(* Logix 5000 project; controller R5_CSS vendor 1 type 14 code 74 rev 19.11; software revision 19.01; part 3 of 20 *)
(* tags used below, declared in another part *)
   AT102A_SCP : SCLP;   // QUENCH WATER CONDUCTIVITY TRANSMITTER SCALER (0-100 milli Siemens)
   AC102A : ANALYTICAL;   // QUENCH WATER CONDUCTIVITY CONTROL
   AlarmMaster : DINT;
   Coal_Tank_Heel_Inches : REAL;
   FC215 : FLOW_CONTROL;   // OVERHEAD CONDENSER CHILLED WATER FLOW CONTROL
   FC365 : FLOW_CONTROL;   // COALESCER PROCESS IMPURITY FLOW CONTROL
   FC370 : FLOW_CONTROL;   // COALESCER MAKE UP WATER FLOW CONTROL
   FC406 : FLOW_CONTROL;   // HX COOLING WATER FLOW CONTROL
   FC_215SCP : SCLP;   // OVERHEAD CONDENSER CHILLED WATER FLOW TRANSMITTER SCALER
   FC_406SCP : SCLP;   // HX COOLING WATER FLOW TRANMITTER SCALER
   FCV410_Open : BOOL;
   FIT08 : BOOL;
   FIT101 : BOOL;
   FIT140A : BOOL;
   FIT140B : BOOL;
   FIT365_SCP : SCLP;   // COALESCER PROCESS IMPURITY FLOW
   FIT370_SCP : SCLP;   // COALESCER MAKE UP WATER SCALER
   FIT403 : BOOL;
   HCP_FAULT : BOOL;
   HS104A : ValveControl_TwoWay;
   HS104B : ValveControl_TwoWay;
   HS141 : ValveControl_TwoWay;
   HS315A : ValveControl_TwoWay;
   HS315B : ValveControl_TwoWay;
   HS431A : ValveControl_TwoWay;
   HS431B : ValveControl_TwoWay;
   HS433A : ValveControl_TwoWay;
   HS433B : ValveControl_TwoWay;
   HT_FAULT : BOOL;
   HTGA : BOOL;
   HX401A : PUMP_CONTROL;   // HEAT EXCHANGER A
   HX401B : PUMP_CONTROL;   // HEAT EXCHANGER B
   InputMax_IF8 : REAL;
   InputMin_IF8 : REAL;
   LC205 : LEVEL_CONTROL;   // OVERHEAD CONDENSER BASIN LEVEL CONTROL
   LC302 : LEVEL_CONTROL;   // COALESCER OIL CHAMBER LEVEL CONTROL
   LC302_LT_Raw : REAL;
   LC302_SP : SCLP;   // COALESCER OIL CHAMBER LEVEL TRANSMITTER SCALER
   LC_205_SCP : SCLP;   // OVERHEAD CONDENSER BASIN LEVEL TRANSMITTER SCALER
   LossOfSignal_mA : DINT;
   MV361_Open : BOOL;
   P101A : PUMP_CONTROL;
   P101B : PUMP_CONTROL;
   P205 : PUMP_CONTROL;   // OVERHEAD CONDENSER TRANSFER PUMP
   P302A : PUMP_CONTROL;
   P302B : PUMP_CONTROL;
   P303A : PUMP_CONTROL;
   P303B : PUMP_CONTROL;
   PC101A : PRESSURE_CONTROL;   // LOWER QUENCH TOWER PRESSURE TRANSMITTER
   PC101B : PRESSURE_CONTROL;   // UPPER QUENCH TOWER PRESSURE TRANSMITTER PRESSURE CONTOL
   PC102A : PRESSURE_CONTROL;   // QUENCH BASIN TRANSFER PUMP SUCTION PRESSURE CONTROL
   PC102B : PRESSURE_CONTROL;   // QUENCH BASIN TRANSFER PUMP DISCHARGE PRESSURE CONTROL
   PC214 : PRESSURE_CONTROL;   // VACUUM SYSTEM PRESSURE TRANSMITTER
   PC214_PID_PV_Select : DINT;   // 0 = PT214 1 = PT101A 2 = PT101B
   PC214_SCP : SCLP;   // VACUUM SYSTEM PRESSURE TRANSMITTER SCALER
   PC271 : PRESSURE_CONTROL;   // VENT HEADER PRESSURE CONTROL
   PC407A : PRESSURE_CONTROL;   // PRE HX LOW PRESSURE TRANSMITTER
   PC407B : PRESSURE_CONTROL;   // POST HX LOW PRESSURE TRANSMITTER
   PIT101A_SCP : SCLP;   // LOWER QUENCH TOWER PRESSURE TRANSMITTER SCALER
   PIT101B_SCP : SCLP;   // UPPER QUENCH TOWER PRESSURE TRANSMITTER SCALER
   PIT102A_SCP : SCLP;   // QUENCH BASIN TRANSFER PUMP SUCTION PRESSURE INDICATOR SCALER
   PIT102B_SCP : SCLP;   // QUENCH BASIN TRANSFER PUMP DISCHARGE PRESSURE SCALER
   PIT407A_SCP : SCLP;   // PRE HX LOW PRESSURE TRANSMITTER
   PIT407B_SCP : SCLP;   // POST HX LOW PRESSURE TRANSMITTER SCALER
   PT271_SCP : SCLP;   // VENT HEADER PRESSURE TRANSMITTER SCALER
   SignalLossHigh_IF8 : DINT;
   SignalLossLow_IF8 : DINT;
   TAS15569 : BOOL;
   TC108 : TEMP_CONTROL;   // QUENCH TOWER EXIT GAS TEMPERATURE CONTROL
   TC114A : TEMP_CONTROL;   // QUENCH BASIN SHELL TEMPERATURE CONTROL
   TC114B : TEMP_CONTROL;   // QUENCH BASIN LIQUID TEMPERATURE CONTROL
   TC121A : TEMP_CONTROL;   // GTL FROM PRUA TEMPERATURE CONTROL
   TC121B : TEMP_CONTROL;   // GTL FROM PRUB TEMPERATURE CONTROL
   TC121C : TEMP_CONTROL;   // GTL FROM PRUC TEMPERATURE CONTROL
   TC121D : TEMP_CONTROL;   // GTL FROM PRUD TEMPERATURE CONTROL
   TC121E : TEMP_CONTROL;
   TC121F : TEMP_CONTROL;
   TC121G : TEMP_CONTROL;
   TC121H : TEMP_CONTROL;
   TC123A : TEMP_CONTROL;   // HEAT JACKET VENT FROM PRUA TEMPERATURE CONTROL
   TC123A_SCP : SCLP;   // HEAT JACKET VENT FROM PRUA TEMPERATURE TRANSMITTER SCALER
   TC123B : TEMP_CONTROL;
   TC123B_SCP : SCLP;   // HEAT JACKET VENT FROM PRUB TEMPERATURE TRANSMITTER SCALER
   TC123C : TEMP_CONTROL;   // HEAT JACKET VENT FROM PRUC TEMPERATURE CONTROL
   TC123C_SCP : SCLP;   // HEAT JACKET VENT FROM PRUC TEMPERATURE TRANSMITTER SCALER
   TC123D : TEMP_CONTROL;   // HEAT JACKET VENT FROM PRUD TEMPERATURE TRANSMITTER
   TC123D_SCP : SCLP;   // HEAT JACKET VENT FROM PRUD TEMPERATURE TRANSMITTER SCALER
   TC123E : TEMP_CONTROL;
   TC123E_SCP : SCLP;
   TC123F : TEMP_CONTROL;
   TC123F_SCP : SCLP;
   TC123G : TEMP_CONTROL;
   TC123G_SCP : SCLP;
   TC306 : TEMP_CONTROL;
   TC313A : TEMP_CONTROL;   // PRIMARY COALESCER SEPARATOR TEMPERATURE CONTROL
   TC319 : TEMP_CONTROL;   // COALESCER OIL CHAMBER PROCESS TEMPERATURE CONTROL
   TT108_SCP : SCLP;   // QUENCH TOWER EXIT GAS TEMPERATURE TRANSMITTER SCALER
   TT121A_SCP : SCLP;   // GTL FROM PRUA TEMPERATURE TRANSMITTER SCALER
   TT121B_SCP : SCLP;
   TT121C_SCP : SCLP;
   TT121D_SCP : SCLP;
   TT121E_SCP : SCLP;
   TT121F_SCP : SCLP;   // GTL FROM PRUB TEMPERATURE TRANSMITTER SCALER
   TT121G_SCP : SCLP;   // GTL FROM PRUC TEMPERATURE TRANSMITTER SCALER
   TT121H_SCP : SCLP;   // GTL FROM PRUD TEMPERATURE TRANSMITTER SCALER
(* MainProgram, continued *)

ROUTINE A1c_MDI   (* ladder *)
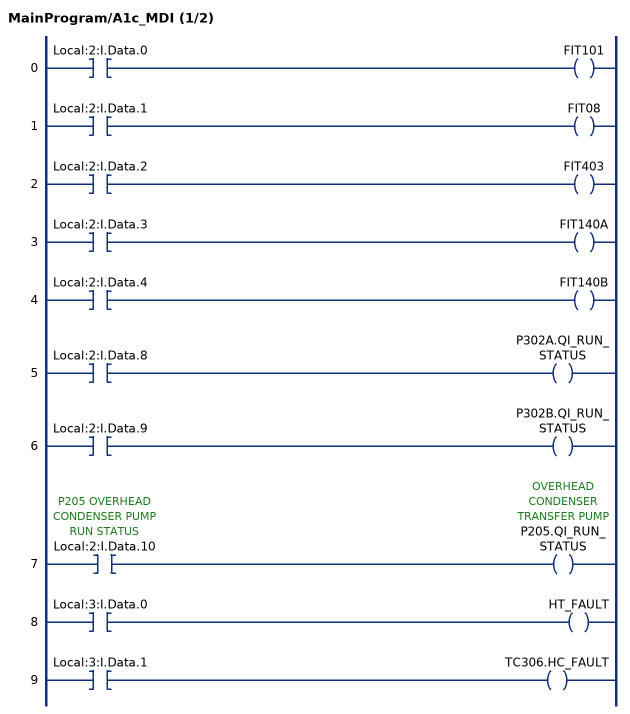
   0: XIC(Local:2:I.Data.0)OTE(FIT101);
   1: XIC(Local:2:I.Data.1)OTE(FIT08);
   2: XIC(Local:2:I.Data.2)OTE(FIT403);
   3: XIC(Local:2:I.Data.3)OTE(FIT140A);
   4: XIC(Local:2:I.Data.4)OTE(FIT140B);
   5: XIC(Local:2:I.Data.8)OTE(P302A.QI_RUN_STATUS);
   6: XIC(Local:2:I.Data.9)OTE(P302B.QI_RUN_STATUS);
   7: XIC(Local:2:I.Data.10)OTE(P205.QI_RUN_STATUS);
   8: XIC(Local:3:I.Data.0)OTE(HT_FAULT);
   9: XIC(Local:3:I.Data.1)OTE(TC306.HC_FAULT);
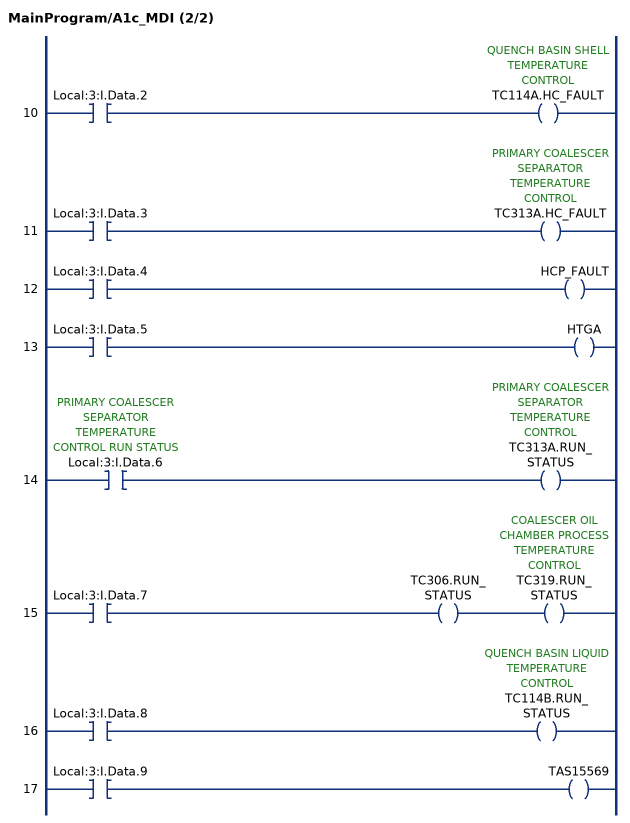
   10: XIC(Local:3:I.Data.2)OTE(TC114A.HC_FAULT);
   11: XIC(Local:3:I.Data.3)OTE(TC313A.HC_FAULT);
   12: XIC(Local:3:I.Data.4)OTE(HCP_FAULT);
   13: XIC(Local:3:I.Data.5)OTE(HTGA);
   14: XIC(Local:3:I.Data.6)OTE(TC313A.RUN_STATUS);
   15: XIC(Local:3:I.Data.7)OTE(TC306.RUN_STATUS)OTE(TC319.RUN_STATUS);
   16: XIC(Local:3:I.Data.8)OTE(TC114B.RUN_STATUS);
   17: XIC(Local:3:I.Data.9)OTE(TAS15569);
END_ROUTINE

ROUTINE A1d_MDO   (* ladder *)
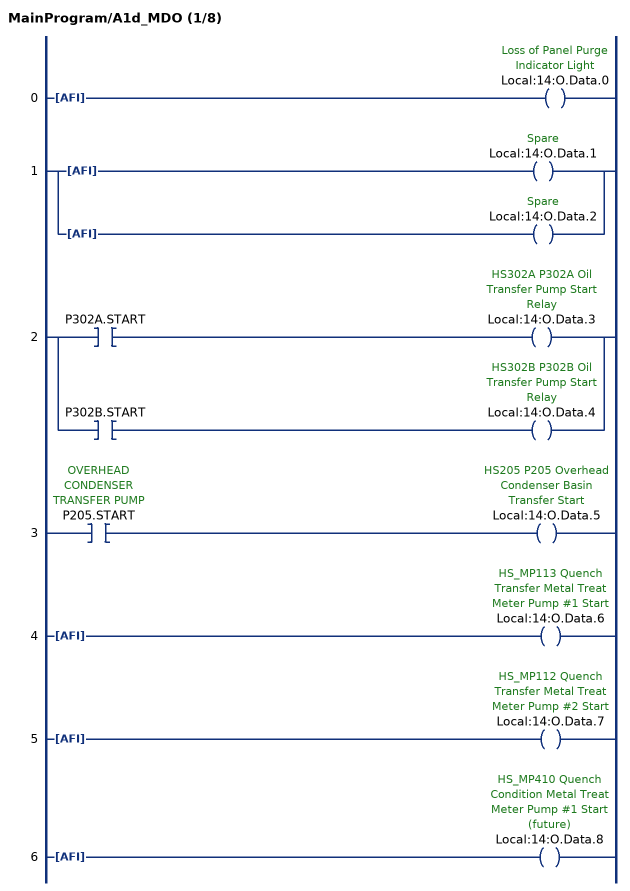
   0: AFI()OTE(Local:14:O.Data.0);
   1: [AFI() OTE(Local:14:O.Data.1) ,AFI() OTE(Local:14:O.Data.2) ];
   2: [XIC(P302A.START) OTE(Local:14:O.Data.3) ,XIC(P302B.START) OTE(Local:14:O.Data.4) ];
   3: XIC(P205.START)OTE(Local:14:O.Data.5);
   4: AFI()OTE(Local:14:O.Data.6);
   5: AFI()OTE(Local:14:O.Data.7);
   6: AFI()OTE(Local:14:O.Data.8);
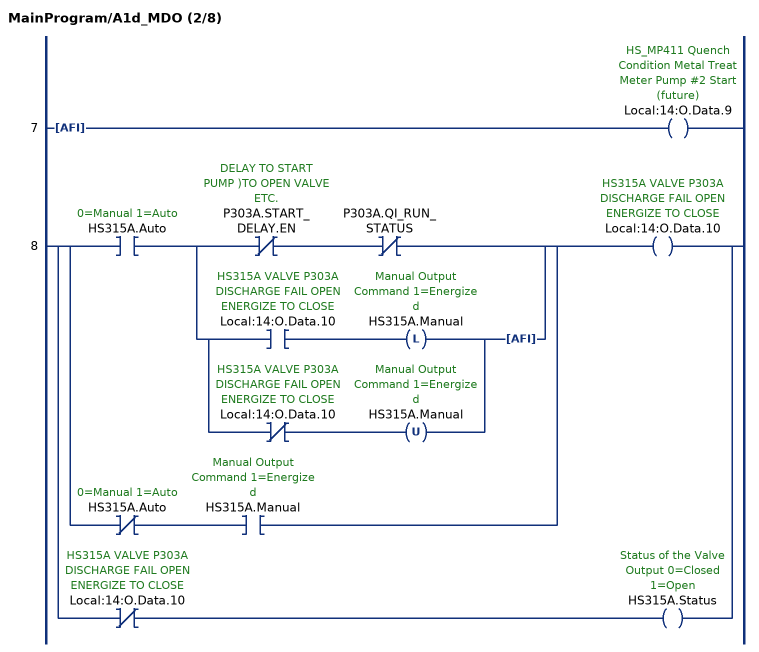
   7: AFI()OTE(Local:14:O.Data.9);
   8: [[XIC(HS315A.Auto) [XIO(P303A.START_DELAY.EN) XIO(P303A.QI_RUN_STATUS) ,[XIC(Local:14:O.Data.10) OTL(HS315A.Manual) ,XIO(Local:14:O.Data.10) OTU(HS315A.Manual) ] AFI() ] ,XIO(HS315A.Auto) XIC(HS315A.Manual) ] OTE(Local:14:O.Data.10) ,XIO(Local:14:O.Data.10) OTE(HS315A.Status) ];
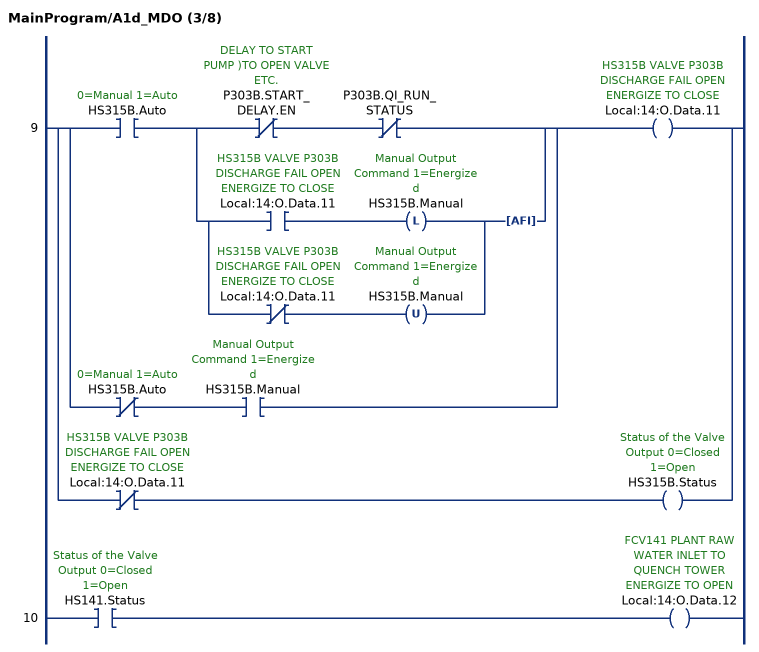
   9: [[XIC(HS315B.Auto) [XIO(P303B.START_DELAY.EN) XIO(P303B.QI_RUN_STATUS) ,[XIC(Local:14:O.Data.11) OTL(HS315B.Manual) ,XIO(Local:14:O.Data.11) OTU(HS315B.Manual) ] AFI() ] ,XIO(HS315B.Auto) XIC(HS315B.Manual) ] OTE(Local:14:O.Data.11) ,XIO(Local:14:O.Data.11) OTE(HS315B.Status) ];
   10: XIC(HS141.Status)OTE(Local:14:O.Data.12);
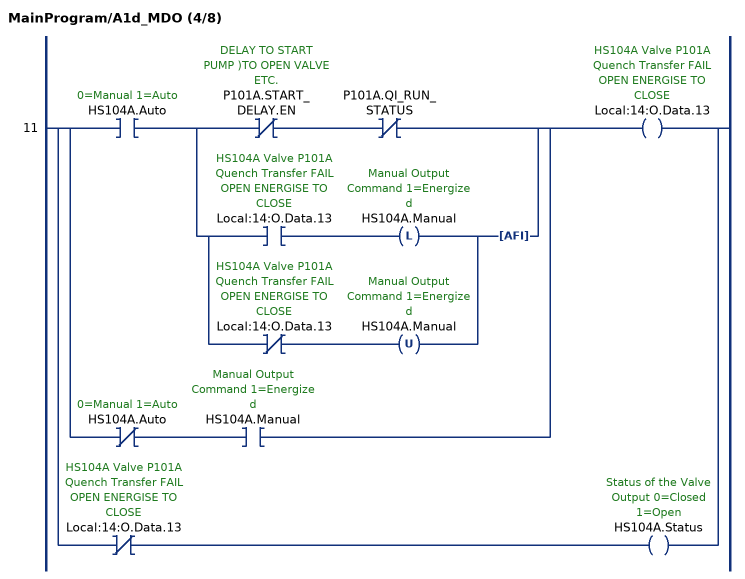
   11: [[XIC(HS104A.Auto) [XIO(P101A.START_DELAY.EN) XIO(P101A.QI_RUN_STATUS) ,[XIC(Local:14:O.Data.13) OTL(HS104A.Manual) ,XIO(Local:14:O.Data.13) OTU(HS104A.Manual) ] AFI() ] ,XIO(HS104A.Auto) XIC(HS104A.Manual) ] OTE(Local:14:O.Data.13) ,XIO(Local:14:O.Data.13) OTE(HS104A.Status) ];
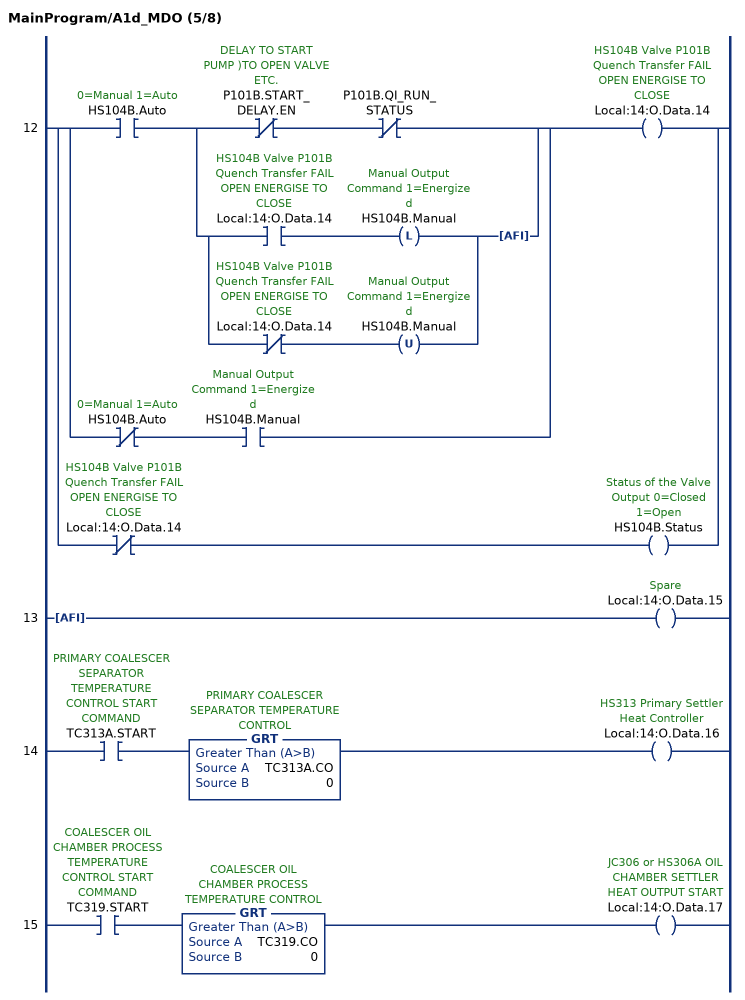
   12: [[XIC(HS104B.Auto) [XIO(P101B.START_DELAY.EN) XIO(P101B.QI_RUN_STATUS) ,[XIC(Local:14:O.Data.14) OTL(HS104B.Manual) ,XIO(Local:14:O.Data.14) OTU(HS104B.Manual) ] AFI() ] ,XIO(HS104B.Auto) XIC(HS104B.Manual) ] OTE(Local:14:O.Data.14) ,XIO(Local:14:O.Data.14) OTE(HS104B.Status) ];
   13: AFI()OTE(Local:14:O.Data.15);
   14: XIC(TC313A.START)GRT(TC313A.CO,0)OTE(Local:14:O.Data.16);
   15: XIC(TC319.START)GRT(TC319.CO,0)OTE(Local:14:O.Data.17);
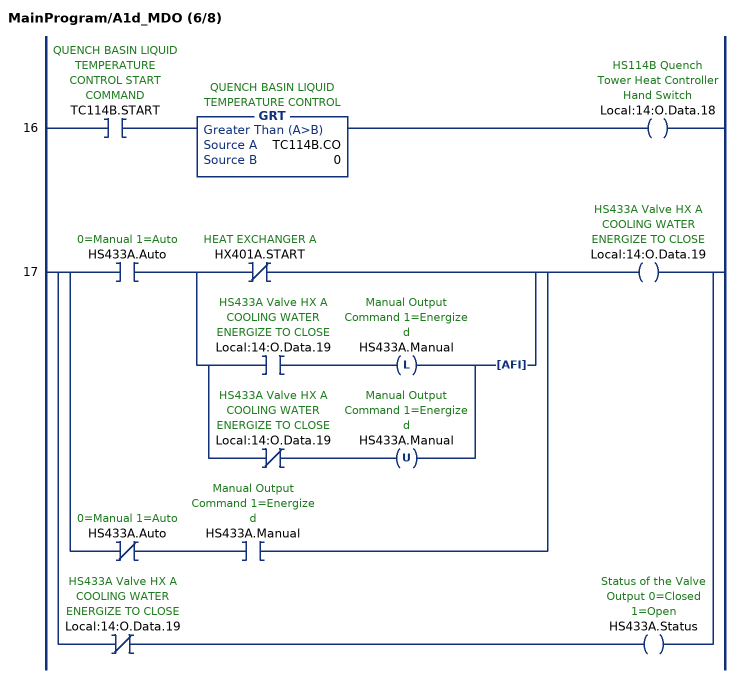
   16: XIC(TC114B.START)GRT(TC114B.CO,0)OTE(Local:14:O.Data.18);
   17: [[XIC(HS433A.Auto) [XIO(HX401A.START) ,[XIC(Local:14:O.Data.19) OTL(HS433A.Manual) ,XIO(Local:14:O.Data.19) OTU(HS433A.Manual) ] AFI() ] ,XIO(HS433A.Auto) XIC(HS433A.Manual) ] OTE(Local:14:O.Data.19) ,XIO(Local:14:O.Data.19) OTE(HS433A.Status) ];
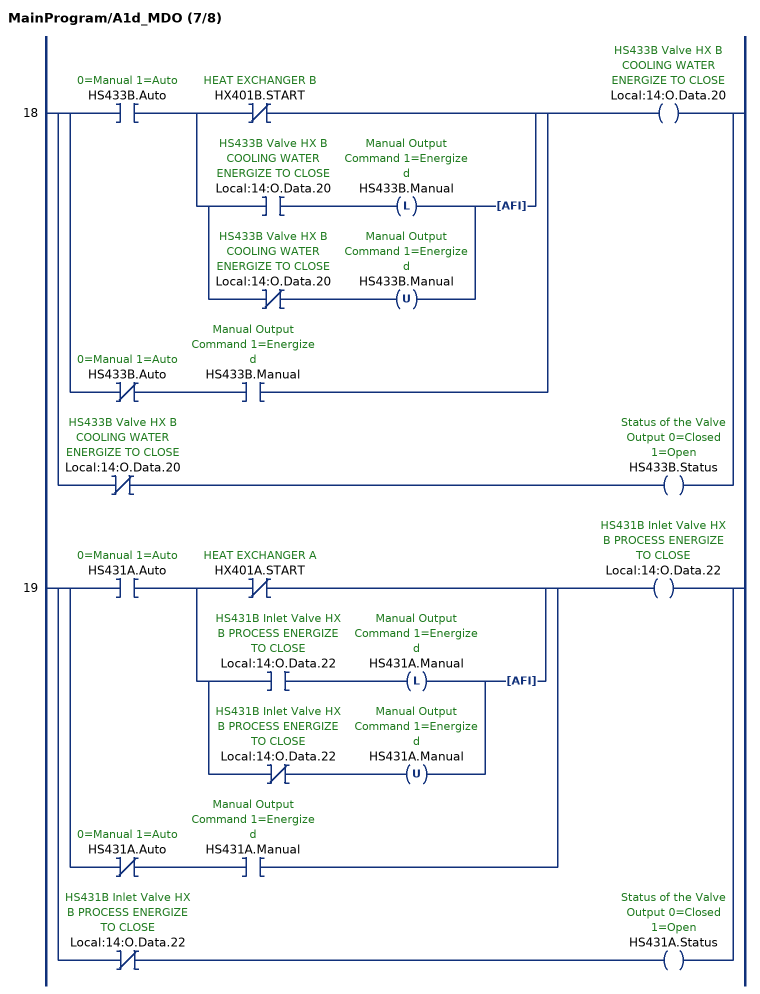
   18: [[XIC(HS433B.Auto) [XIO(HX401B.START) ,[XIC(Local:14:O.Data.20) OTL(HS433B.Manual) ,XIO(Local:14:O.Data.20) OTU(HS433B.Manual) ] AFI() ] ,XIO(HS433B.Auto) XIC(HS433B.Manual) ] OTE(Local:14:O.Data.20) ,XIO(Local:14:O.Data.20) OTE(HS433B.Status) ];
   19: [[XIC(HS431A.Auto) [XIO(HX401A.START) ,[XIC(Local:14:O.Data.22) OTL(HS431A.Manual) ,XIO(Local:14:O.Data.22) OTU(HS431A.Manual) ] AFI() ] ,XIO(HS431A.Auto) XIC(HS431A.Manual) ] OTE(Local:14:O.Data.22) ,XIO(Local:14:O.Data.22) OTE(HS431A.Status) ];
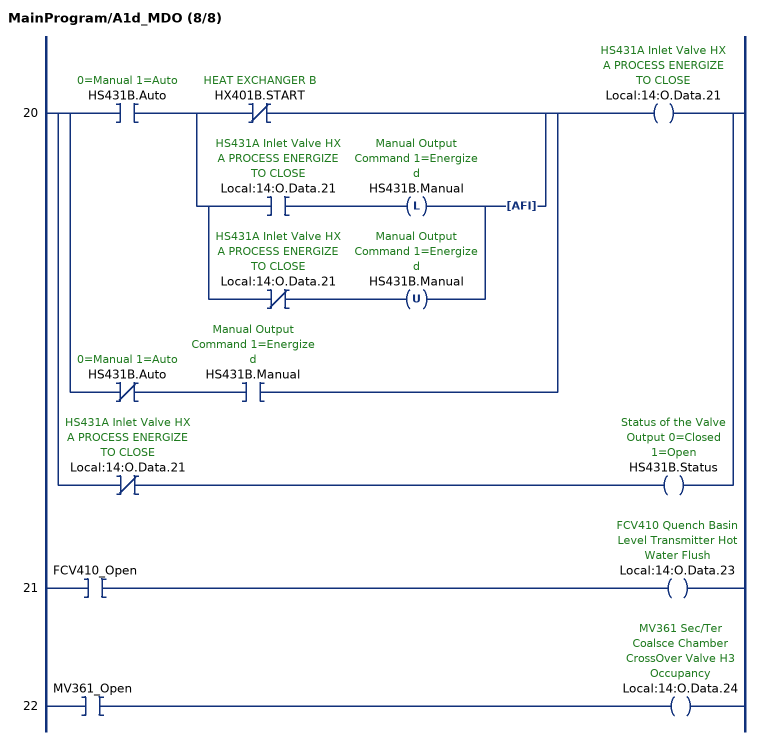
   20: [[XIC(HS431B.Auto) [XIO(HX401B.START) ,[XIC(Local:14:O.Data.21) OTL(HS431B.Manual) ,XIO(Local:14:O.Data.21) OTU(HS431B.Manual) ] AFI() ] ,XIO(HS431B.Auto) XIC(HS431B.Manual) ] OTE(Local:14:O.Data.21) ,XIO(Local:14:O.Data.21) OTE(HS431B.Status) ];
   21: XIC(FCV410_Open)OTE(Local:14:O.Data.23);
   22: XIC(MV361_Open)OTE(Local:14:O.Data.24);
END_ROUTINE

ROUTINE A1e_MAI_SCP   (* ladder *)
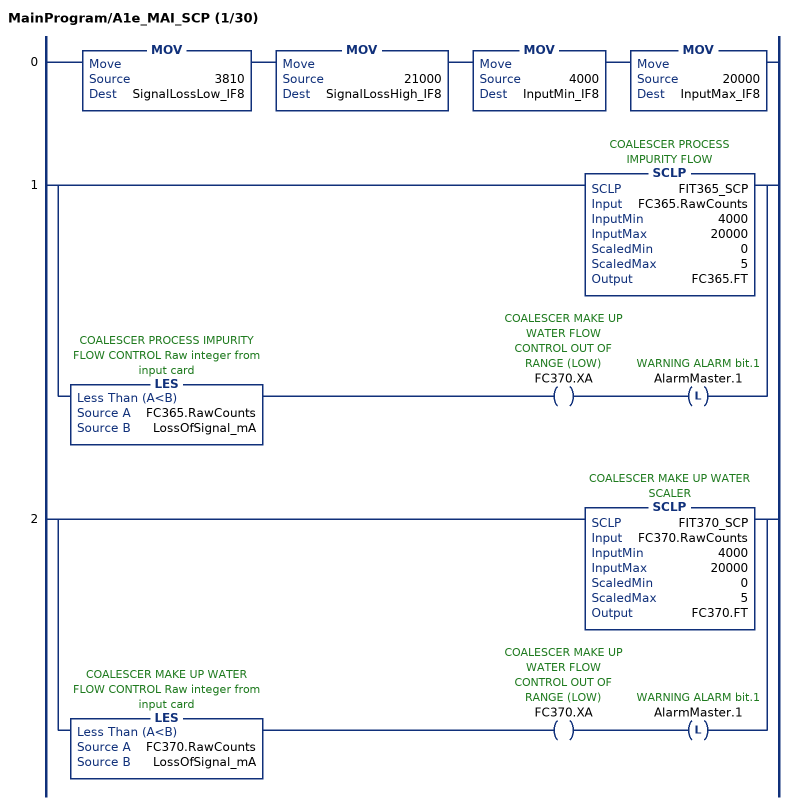
   0: MOV(3810,SignalLossLow_IF8)MOV(21000,SignalLossHigh_IF8)MOV(4000,InputMin_IF8)MOV(20000,InputMax_IF8);
   1: [SCLP(FIT365_SCP,FC365.RawCounts,4000,20000,0,5,FC365.FT) ,LES(FC365.RawCounts,LossOfSignal_mA) OTE(FC370.XA) OTL(AlarmMaster.1) ];
   2: [SCLP(FIT370_SCP,FC370.RawCounts,4000,20000,0,5,FC370.FT) ,LES(FC370.RawCounts,LossOfSignal_mA) OTE(FC370.XA) OTL(AlarmMaster.1) ];
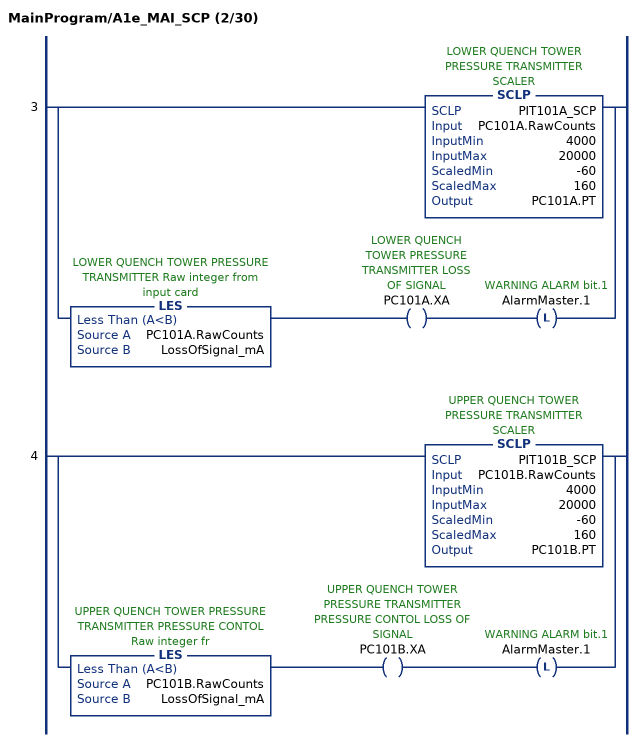
   3: [SCLP(PIT101A_SCP,PC101A.RawCounts,4000,20000,-60,160,PC101A.PT) ,LES(PC101A.RawCounts,LossOfSignal_mA) OTE(PC101A.XA) OTL(AlarmMaster.1) ];
   4: [SCLP(PIT101B_SCP,PC101B.RawCounts,4000,20000,-60,160,PC101B.PT) ,LES(PC101B.RawCounts,LossOfSignal_mA) OTE(PC101B.XA) OTL(AlarmMaster.1) ];
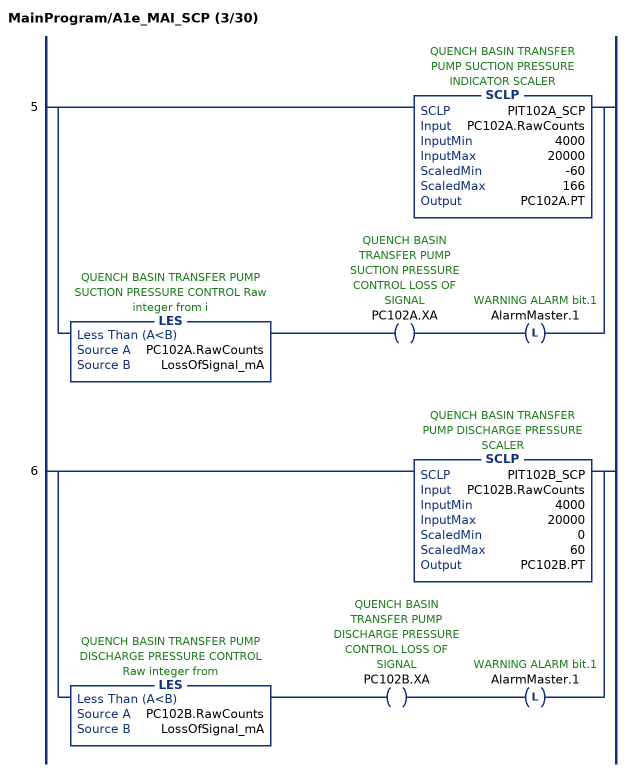
   5: [SCLP(PIT102A_SCP,PC102A.RawCounts,4000,20000,-60,166,PC102A.PT) ,LES(PC102A.RawCounts,LossOfSignal_mA) OTE(PC102A.XA) OTL(AlarmMaster.1) ];
   6: [SCLP(PIT102B_SCP,PC102B.RawCounts,4000,20000,0,60,PC102B.PT) ,LES(PC102B.RawCounts,LossOfSignal_mA) OTE(PC102B.XA) OTL(AlarmMaster.1) ];
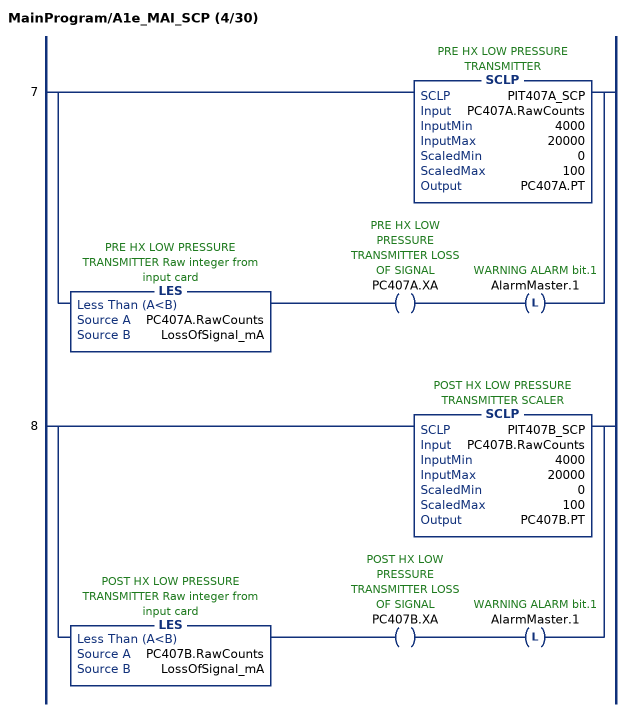
   7: [SCLP(PIT407A_SCP,PC407A.RawCounts,4000,20000,0,100,PC407A.PT) ,LES(PC407A.RawCounts,LossOfSignal_mA) OTE(PC407A.XA) OTL(AlarmMaster.1) ];
   8: [SCLP(PIT407B_SCP,PC407B.RawCounts,4000,20000,0,100,PC407B.PT) ,LES(PC407B.RawCounts,LossOfSignal_mA) OTE(PC407B.XA) OTL(AlarmMaster.1) ];
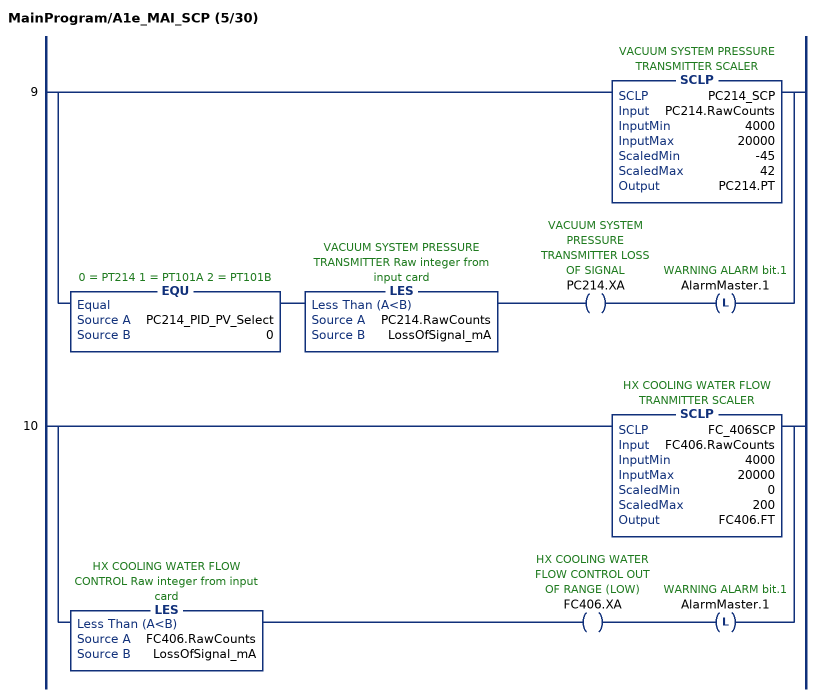
   9: [SCLP(PC214_SCP,PC214.RawCounts,4000,20000,-45,42,PC214.PT) ,EQU(PC214_PID_PV_Select,0) LES(PC214.RawCounts,LossOfSignal_mA) OTE(PC214.XA) OTL(AlarmMaster.1) ];
   10: [SCLP(FC_406SCP,FC406.RawCounts,4000,20000,0,200,FC406.FT) ,LES(FC406.RawCounts,LossOfSignal_mA) OTE(FC406.XA) OTL(AlarmMaster.1) ];
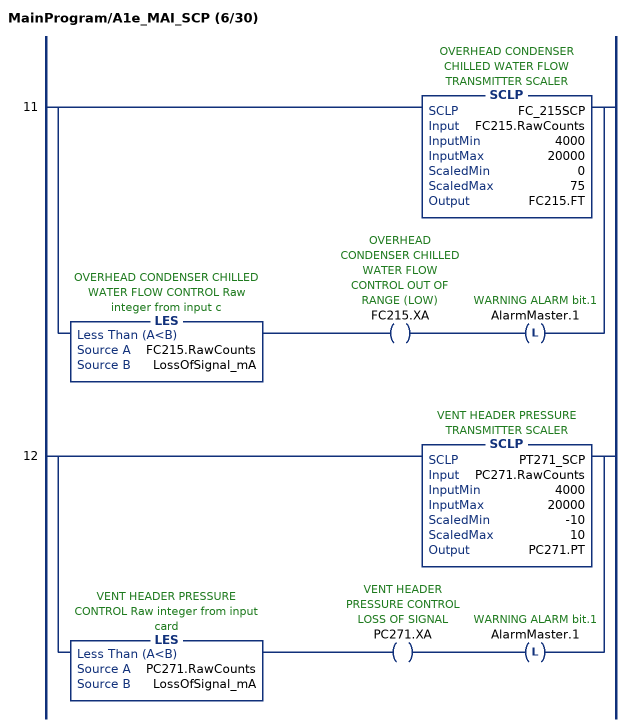
   11: [SCLP(FC_215SCP,FC215.RawCounts,4000,20000,0,75,FC215.FT) ,LES(FC215.RawCounts,LossOfSignal_mA) OTE(FC215.XA) OTL(AlarmMaster.1) ];
   12: [SCLP(PT271_SCP,PC271.RawCounts,4000,20000,-10,10,PC271.PT) ,LES(PC271.RawCounts,LossOfSignal_mA) OTE(PC271.XA) OTL(AlarmMaster.1) ];
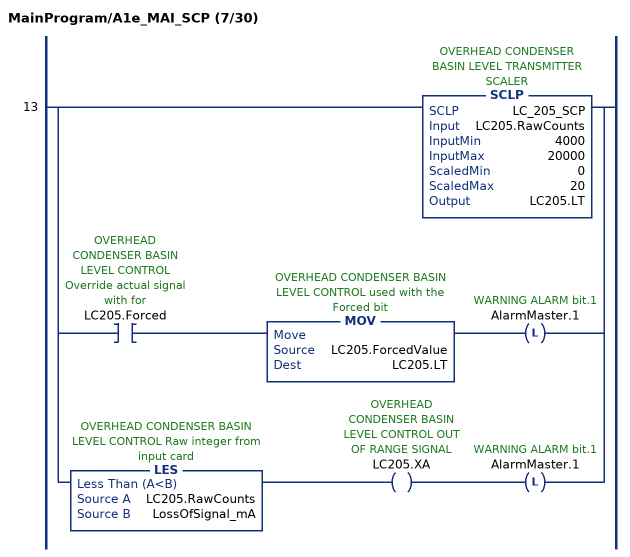
   13: [SCLP(LC_205_SCP,LC205.RawCounts,4000,20000,0,20,LC205.LT) ,XIC(LC205.Forced) MOV(LC205.ForcedValue,LC205.LT) OTL(AlarmMaster.1) ,LES(LC205.RawCounts,LossOfSignal_mA) OTE(LC205.XA) OTL(AlarmMaster.1) ];
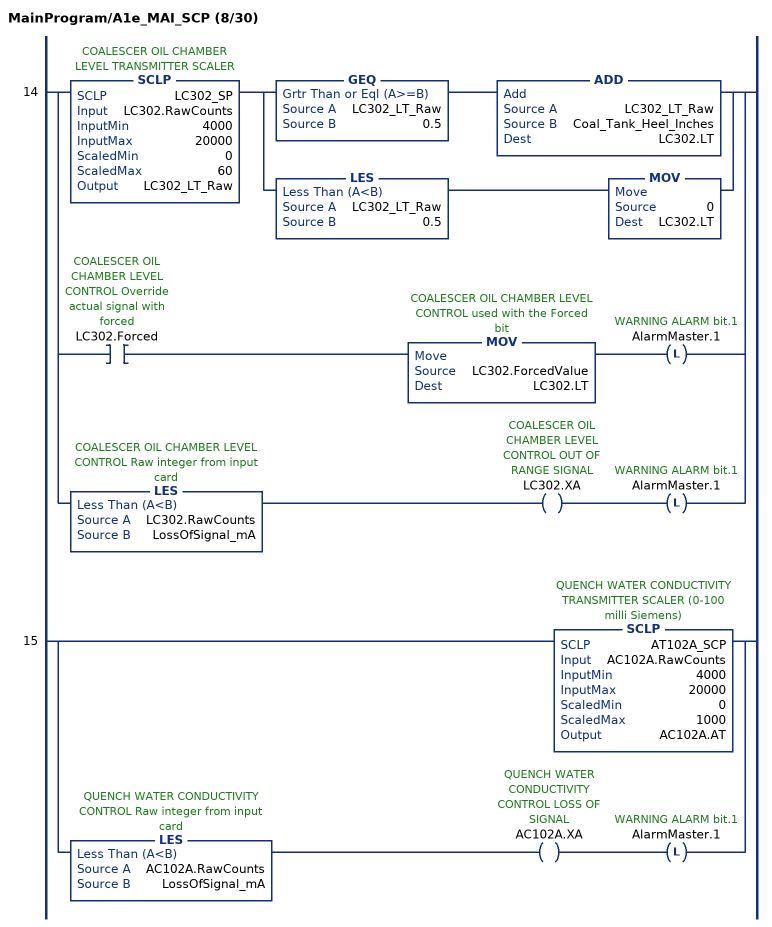
   14: [SCLP(LC302_SP,LC302.RawCounts,4000,20000,0,60,LC302_LT_Raw) [GEQ(LC302_LT_Raw,0.5) ADD(LC302_LT_Raw,Coal_Tank_Heel_Inches,LC302.LT) ,LES(LC302_LT_Raw,0.5) MOV(0,LC302.LT) ] ,XIC(LC302.Forced) MOV(LC302.ForcedValue,LC302.LT) OTL(AlarmMaster.1) ,LES(LC302.RawCounts,LossOfSignal_mA) OTE(LC302.XA) OTL(AlarmMaster.1) ];
   15: [SCLP(AT102A_SCP,AC102A.RawCounts,4000,20000,0,1000,AC102A.AT) ,LES(AC102A.RawCounts,LossOfSignal_mA) OTE(AC102A.XA) OTL(AlarmMaster.1) ];
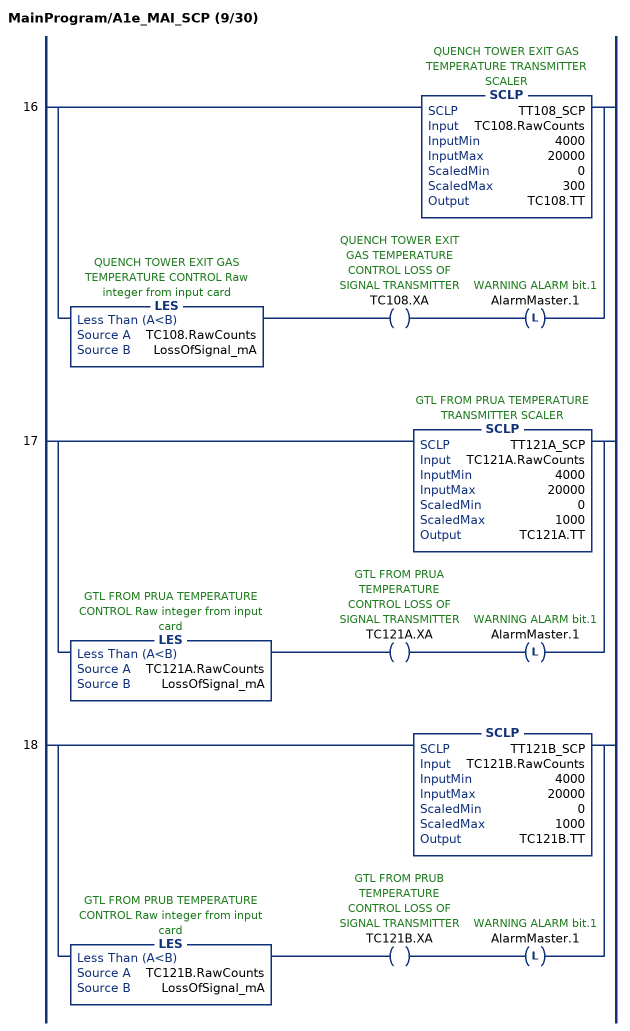
   16: [SCLP(TT108_SCP,TC108.RawCounts,4000,20000,0,300,TC108.TT) ,LES(TC108.RawCounts,LossOfSignal_mA) OTE(TC108.XA) OTL(AlarmMaster.1) ];
   17: [SCLP(TT121A_SCP,TC121A.RawCounts,4000,20000,0,1000,TC121A.TT) ,LES(TC121A.RawCounts,LossOfSignal_mA) OTE(TC121A.XA) OTL(AlarmMaster.1) ];
   18: [SCLP(TT121B_SCP,TC121B.RawCounts,4000,20000,0,1000,TC121B.TT) ,LES(TC121B.RawCounts,LossOfSignal_mA) OTE(TC121B.XA) OTL(AlarmMaster.1) ];
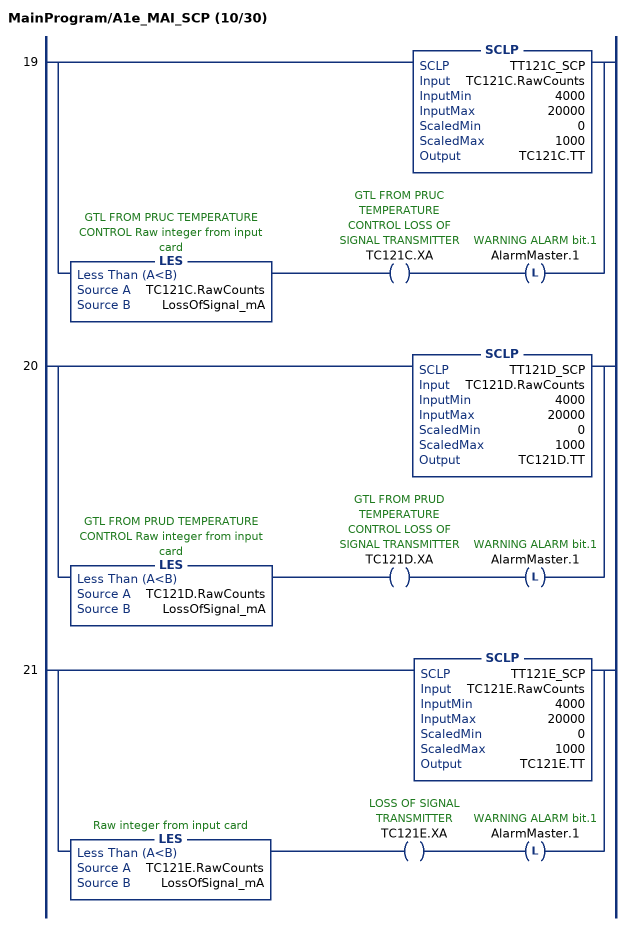
   19: [SCLP(TT121C_SCP,TC121C.RawCounts,4000,20000,0,1000,TC121C.TT) ,LES(TC121C.RawCounts,LossOfSignal_mA) OTE(TC121C.XA) OTL(AlarmMaster.1) ];
   20: [SCLP(TT121D_SCP,TC121D.RawCounts,4000,20000,0,1000,TC121D.TT) ,LES(TC121D.RawCounts,LossOfSignal_mA) OTE(TC121D.XA) OTL(AlarmMaster.1) ];
   21: [SCLP(TT121E_SCP,TC121E.RawCounts,4000,20000,0,1000,TC121E.TT) ,LES(TC121E.RawCounts,LossOfSignal_mA) OTE(TC121E.XA) OTL(AlarmMaster.1) ];
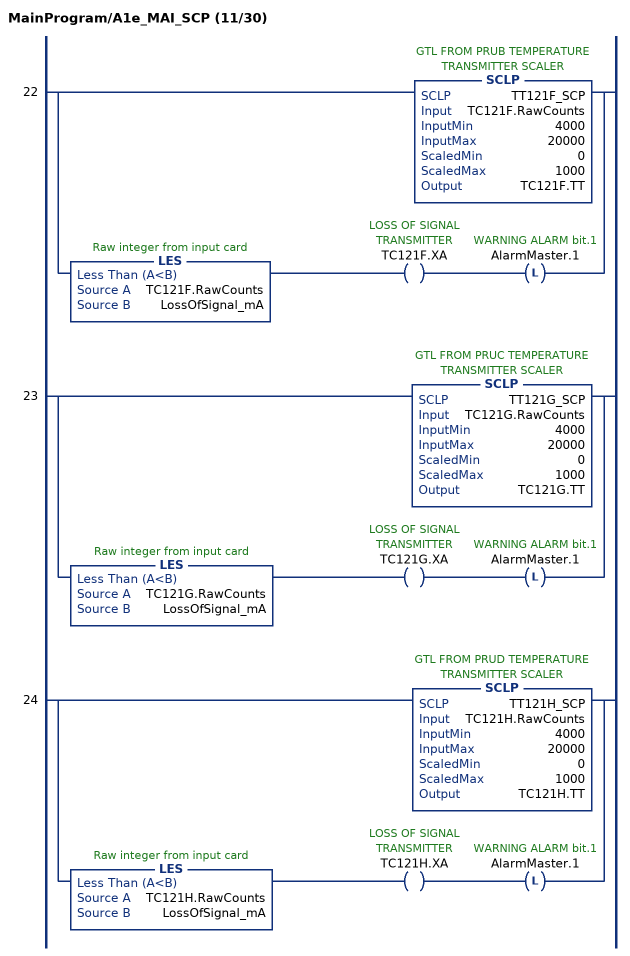
   22: [SCLP(TT121F_SCP,TC121F.RawCounts,4000,20000,0,1000,TC121F.TT) ,LES(TC121F.RawCounts,LossOfSignal_mA) OTE(TC121F.XA) OTL(AlarmMaster.1) ];
   23: [SCLP(TT121G_SCP,TC121G.RawCounts,4000,20000,0,1000,TC121G.TT) ,LES(TC121G.RawCounts,LossOfSignal_mA) OTE(TC121G.XA) OTL(AlarmMaster.1) ];
   24: [SCLP(TT121H_SCP,TC121H.RawCounts,4000,20000,0,1000,TC121H.TT) ,LES(TC121H.RawCounts,LossOfSignal_mA) OTE(TC121H.XA) OTL(AlarmMaster.1) ];
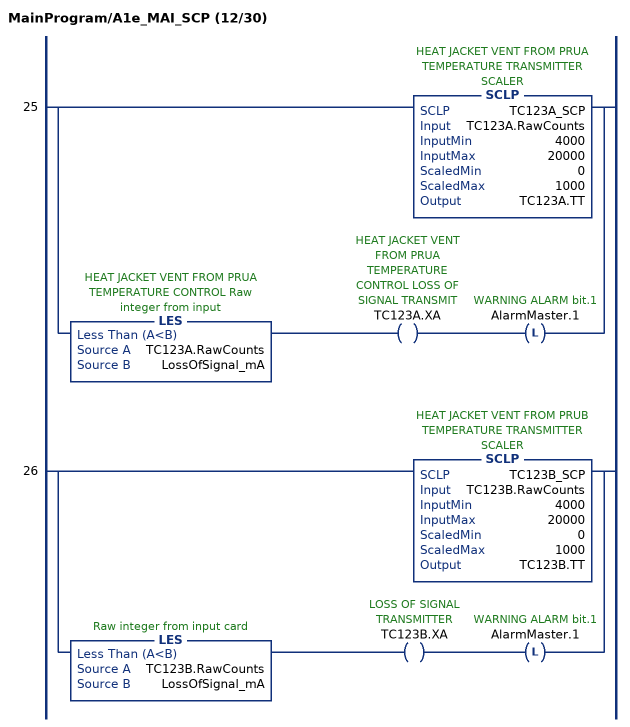
   25: [SCLP(TC123A_SCP,TC123A.RawCounts,4000,20000,0,1000,TC123A.TT) ,LES(TC123A.RawCounts,LossOfSignal_mA) OTE(TC123A.XA) OTL(AlarmMaster.1) ];
   26: [SCLP(TC123B_SCP,TC123B.RawCounts,4000,20000,0,1000,TC123B.TT) ,LES(TC123B.RawCounts,LossOfSignal_mA) OTE(TC123B.XA) OTL(AlarmMaster.1) ];
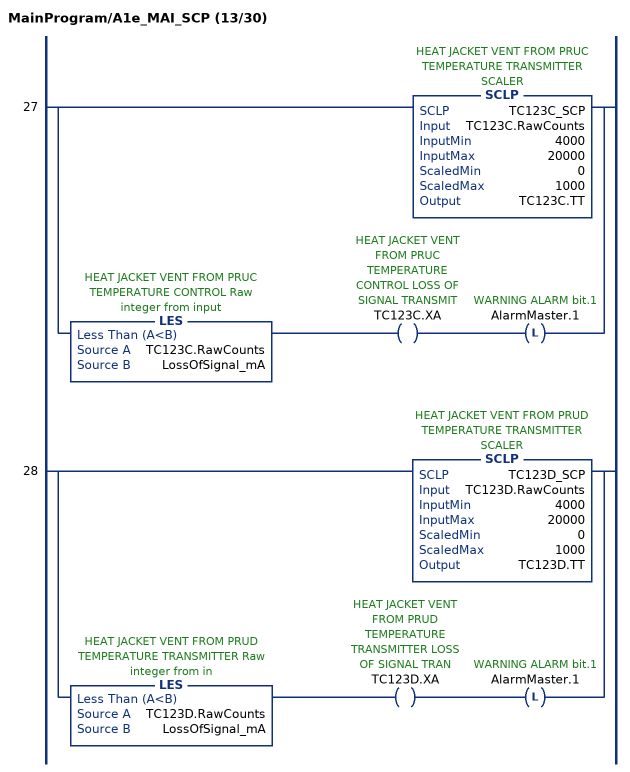
   27: [SCLP(TC123C_SCP,TC123C.RawCounts,4000,20000,0,1000,TC123C.TT) ,LES(TC123C.RawCounts,LossOfSignal_mA) OTE(TC123C.XA) OTL(AlarmMaster.1) ];
   28: [SCLP(TC123D_SCP,TC123D.RawCounts,4000,20000,0,1000,TC123D.TT) ,LES(TC123D.RawCounts,LossOfSignal_mA) OTE(TC123D.XA) OTL(AlarmMaster.1) ];
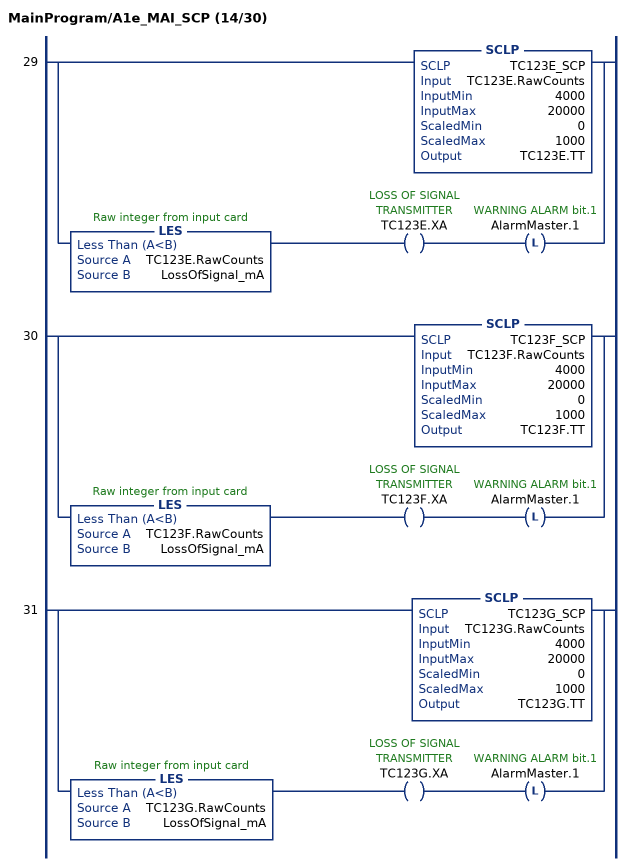
   29: [SCLP(TC123E_SCP,TC123E.RawCounts,4000,20000,0,1000,TC123E.TT) ,LES(TC123E.RawCounts,LossOfSignal_mA) OTE(TC123E.XA) OTL(AlarmMaster.1) ];
   30: [SCLP(TC123F_SCP,TC123F.RawCounts,4000,20000,0,1000,TC123F.TT) ,LES(TC123F.RawCounts,LossOfSignal_mA) OTE(TC123F.XA) OTL(AlarmMaster.1) ];
   31: [SCLP(TC123G_SCP,TC123G.RawCounts,4000,20000,0,1000,TC123G.TT) ,LES(TC123G.RawCounts,LossOfSignal_mA) OTE(TC123G.XA) OTL(AlarmMaster.1) ];
